FUNCTION_BLOCK ArrowheadPublish (* Publish event Function Block *)
  (* Standard: 61499-2; Description: Copyright (c) 2019 fortiss GmbH This program and the accompanying materials are made available under the terms of the Eclipse Public License 2.0 which is available at https://www.eclipse.org/legal/epl-2.0/ SPDX-License-Identifier: EPL-2.0 *)
  (* Version 1.0, 2019-09-17, Cabral, fortiss GmbH *)
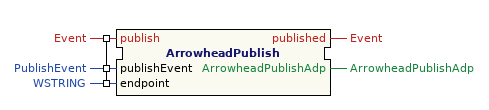
  EVENT_INPUT
    publish WITH publishEvent, endpoint; (* Publish Event *)
  END_EVENT
  EVENT_OUTPUT
    published; (* Event was published *)
  END_EVENT
  VAR_INPUT
    publishEvent : PublishEvent; (* Publish event to be sent *)
    endpoint : WSTRING; (* Endpoint (IP:PORT/URI) of the Event Handler (not officially in the documentation, but it simplifies the FBs) *)
  END_VAR
  PLUGS
    ArrowheadPublishAdp : ArrowheadPublishAdp;
  END_PLUGS
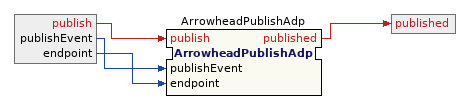
  EVENT_CONNECTIONS
    publish TO ArrowheadPublishAdp.publish;
    ArrowheadPublishAdp.published TO published;
  END_CONNECTIONS
  DATA_CONNECTIONS
    publishEvent TO ArrowheadPublishAdp.publishEvent;
    endpoint TO ArrowheadPublishAdp.endpoint;
  END_CONNECTIONS
END_FUNCTION_BLOCK
